// TwinCAT 3 PLC project OC_TwinCAT_EtherCAT
// Title: OC_EtherCAT
// Company: Open Commissioning
// Author: SpiraTec AG
// ProjectVersion: 1.0.0
// Description: Open Commissioning TwinCAT EtherCAT Library
// ProgramVersion: 3.1.4024.0
// libraries:
//   OC_Core, * (Open Commissioning)
//   Tc2_Standard, * (Beckhoff Automation GmbH)
//   Tc2_System, * (Beckhoff Automation GmbH)
//   Tc3_Module, * (Beckhoff Automation GmbH)
//   TcUnit, * (www.tcunit.org)
// project tree:
//   Devices/FB_Beckhoff_EL6001/ E_Beckhoff_EL6001_State.TcDUT (not stored), FB_Beckhoff_EL6001.TcPOU
//   DUTs/ ST_Baumer_Encoder.TcDUT (not stored), ST_Beckhoff_4AI.TcDUT, ST_Beckhoff_2AI.TcDUT, ST_Beckhoff_EL3403.TcDUT, ST_Beckhoff_EL5002.TcDUT, ST_CoE402.TcDUT, ST_Beckhoff_EL9110.TcDUT, ST_Beckhoff_EL9410.TcDUT, ST_Beckhoff_16DI.TcDUT (not stored), ST_Beckhoff_16DO.TcDUT, ST_Beckhoff_4AO.TcDUT (not stored), ST_Beckhoff_4DI_4DO.TcDUT, ST_Beckhoff_8DI.TcDUT (not stored), ST_Beckhoff_8DI_8DO.TcDUT, ST_Beckhoff_8DO.TcDUT, ST_Gefran_GFX4.TcDUT, ST_SEW_SimMovitrac.TcDUT
//   Devices/ FB_Beckhoff_EL5152.TcPOU
//   / PlcTask.TcTTO
//   Tests/Devices/ FB_Beckhoff_EL5152_Test.TcPOU, FB_Beckhoff_EL6001_Test.TcPOU
//   Tests/ PRG_TEST.TcPOU

CONFIGURATION OC_TwinCAT_EtherCAT
    RESOURCE PLC ON TwinCAT3
        TASK PlcTask(INTERVAL := T#1ms, PRIORITY := 30);
        PROGRAM PRG_TEST WITH PlcTask : PRG_TEST;
    END_RESOURCE
END_CONFIGURATION

// ---- DUTs/ST_Beckhoff_4AI.TcDUT
{attribute 'pack_mode' := '1'} 
TYPE ST_Beckhoff_4AI :
STRUCT
	nStatus1	AT %Q* : UINT;
	nValue1		AT %Q* : INT;
	nStatus2	AT %Q* : UINT;
	nValue2		AT %Q* : INT;
END_STRUCT
END_TYPE

// ---- DUTs/ST_Beckhoff_2AI.TcDUT
{attribute 'pack_mode' := '1'} 
TYPE ST_Beckhoff_2AI :
STRUCT
	nStatus1	AT %Q* : UINT;
	nValue1		AT %Q* : INT;
	nStatus2	AT %Q* : UINT;
	nValue2		AT %Q* : INT;
	nStatus3	AT %Q* : UINT;
	nValue3		AT %Q* : INT;
	nStatus4	AT %Q* : UINT;
	nValue4		AT %Q* : INT;
END_STRUCT
END_TYPE

// ---- DUTs/ST_Beckhoff_EL3403.TcDUT
TYPE ST_Beckhoff_EL3403 :
STRUCT
	nCurrent1		AT %Q* : UINT;
	nVoltage1		AT %Q* : UINT;
	nActivePower1	AT %Q* : UINT;
	nCurrent2		AT %Q* : UINT;
	nVoltage2		AT %Q* : UINT;
	nActivePower2	AT %Q* : UINT;	
	nCurrent3		AT %Q* : UINT;
	nVoltage3		AT %Q* : UINT;
	nActivePower3	AT %Q* : UINT;
END_STRUCT
END_TYPE

// ---- DUTs/ST_Beckhoff_EL5002.TcDUT
TYPE ST_Beckhoff_EL5002 :
STRUCT
	nStatus1	AT %Q* : UINT;
	nCounter1	AT %Q* : UDINT;	
	nStatus2	AT %Q* : UINT;
	nCounter2	AT %Q* : UDINT;	
END_STRUCT
END_TYPE

// ---- DUTs/ST_CoE402.TcDUT
{attribute 'pack_mode' := '1'} 
TYPE ST_CoE402 :
STRUCT
	nControlWord	AT %I* : UINT;
	nTargetValue	AT %I* : DINT;
	nStatusWord		AT %Q* : UINT;
	nActualValue	AT %Q* : DINT;
END_STRUCT
END_TYPE

// ---- DUTs/ST_Beckhoff_EL9110.TcDUT
{attribute 'pack_mode' := '1'} 
TYPE ST_Beckhoff_EL9110 :
STRUCT
	bPowerOk	AT %Q* : BIT := TRUE;
END_STRUCT
END_TYPE

// ---- DUTs/ST_Beckhoff_EL9410.TcDUT
{attribute 'pack_mode' := '1'} 
TYPE ST_Beckhoff_EL9410 :
STRUCT
	bUsUndervoltage	AT %Q* : BIT;
	bUpUndervoltage	AT %Q* : BIT;
END_STRUCT
END_TYPE

// ---- DUTs/ST_Beckhoff_16DO.TcDUT
{attribute 'pack_mode' := '1'} 
TYPE ST_Beckhoff_16DO :
STRUCT
	bOut1	AT %I* : BIT;
	bOut2	AT %I* : BIT;
	bOut3	AT %I* : BIT;
	bOut4	AT %I* : BIT;
	bOut5	AT %I* : BIT;
	bOut6	AT %I* : BIT;
	bOut7	AT %I* : BIT;
	bOut8	AT %I* : BIT;
	bOut9	AT %I* : BIT;
	bOut10	AT %I* : BIT;
	bOut11	AT %I* : BIT;
	bOut12	AT %I* : BIT;
	bOut13	AT %I* : BIT;
	bOut14	AT %I* : BIT;
	bOut15	AT %I* : BIT;
	bOut16	AT %I* : BIT;
END_STRUCT
END_TYPE

// ---- DUTs/ST_Beckhoff_4DI_4DO.TcDUT
{attribute 'pack_mode' := '1'} 
TYPE ST_Beckhoff_4DI_4DO :
STRUCT
	bIn1	AT %Q* : BIT;
	bIn2	AT %Q* : BIT;
	bIn3	AT %Q* : BIT;
	bIn4	AT %Q* : BIT;	
	bOut1	AT %I* : BIT;
	bOut2	AT %I* : BIT;
	bOut3	AT %I* : BIT;
	bOut4	AT %I* : BIT;	
END_STRUCT
END_TYPE

// ---- DUTs/ST_Beckhoff_8DI_8DO.TcDUT
{attribute 'pack_mode' := '1'} 
TYPE ST_Beckhoff_8DI_8DO :
STRUCT
	bIn1	AT %Q* : BIT;
	bIn2	AT %Q* : BIT;
	bIn3	AT %Q* : BIT;
	bIn4	AT %Q* : BIT;
	bIn5	AT %Q* : BIT;
	bIn6	AT %Q* : BIT;
	bIn7	AT %Q* : BIT;
	bIn8	AT %Q* : BIT;
	bOut1	AT %I* : BIT;
	bOut2	AT %I* : BIT;
	bOut3	AT %I* : BIT;
	bOut4	AT %I* : BIT;
	bOut5	AT %I* : BIT;
	bOut6	AT %I* : BIT;
	bOut7	AT %I* : BIT;
	bOut8	AT %I* : BIT;
END_STRUCT
END_TYPE

// ---- DUTs/ST_Beckhoff_8DO.TcDUT
{attribute 'pack_mode' := '1'} 
TYPE ST_Beckhoff_8DO :
STRUCT
	bOut1	AT %I* : BIT;
	bOut2	AT %I* : BIT;
	bOut3	AT %I* : BIT;
	bOut4	AT %I* : BIT;
	bOut5	AT %I* : BIT;
	bOut6	AT %I* : BIT;
	bOut7	AT %I* : BIT;
	bOut8	AT %I* : BIT;
END_STRUCT
END_TYPE

// ---- DUTs/ST_Gefran_GFX4.TcDUT
{attribute 'pack_mode' := '1'} 
TYPE ST_Gefran_GFX4 :
STRUCT
	nProcessVariable1	AT %Q* : INT;
	nControllerStatus1	AT %Q* : UINT;	
	nOutputPower1		AT %Q* : INT;
	nProcessVariable2	AT %Q* : INT;
	nControllerStatus2	AT %Q* : UINT;	
	nOutputPower2		AT %Q* : INT;
	nProcessVariable3	AT %Q* : INT;
	nControllerStatus3	AT %Q* : UINT;	
	nOutputPower3		AT %Q* : INT;
	nProcessVariable4	AT %Q* : INT;
	nControllerStatus4	AT %Q* : UINT;	
	nOutputPower4		AT %Q* : INT;
	nLocalSetpoint1		AT %I* : INT;
	nLocalSetpoint2		AT %I* : INT;
	nLocalSetpoint3		AT %I* : INT;
	nLocalSetpoint4		AT %I* : INT;
END_STRUCT
END_TYPE

// ---- DUTs/ST_SEW_SimMovitrac.TcDUT
{attribute 'pack_mode' := '1'}
TYPE ST_SEW_SimMovitrac :
STRUCT
	PI1		AT %Q* : WORD;
	PI2		AT %Q* : WORD;
	PI3		AT %Q* : WORD;
	PO1		AT %I* : WORD;
	PO2		AT %I* : WORD;
	PO3		AT %I* : WORD;
END_STRUCT
END_TYPE

// ---- Tests/PRG_TEST.TcPOU
PROGRAM PRG_TEST
VAR	
	FB_System	: FB_System;
	FB_Beckhoff_EL5152_Test : FB_Beckhoff_EL5152_Test;
	FB_Beckhoff_EL6001_Test : FB_Beckhoff_EL6001_Test;
	FB_DS402_FSM_Test : FB_DS402_FSM_Test;	
	FB_DS402_CSP_Test : FB_DS402_CSP_Test; 
	FB_Sercos_FSM_Test : FB_Sercos_FSM_Test;
	FB_Sercos_VC_Test : FB_Sercos_VC_Test;
END_VAR

FB_System();
TcUnit.RUN();

END_PROGRAM

// ---- Tests/Devices/FB_Beckhoff_EL5152_Test.TcPOU
FUNCTION_BLOCK FB_Beckhoff_EL5152_Test EXTENDS TcUnit.FB_TestSuite
VAR
	fbDevice : FB_Beckhoff_EL5152;
	nExpected : UINT;
	nResult : UINT;
END_VAR

TEST('nCounter1');
nExpected := 111;
fbDevice.nValue1 := nExpected;
fbDevice();
nResult := fbDevice.Counter1;
AssertEquals(Expected := nExpected,
             Actual := nResult,
             Message := 'nCounter1 value is not correct');	
TEST_FINISHED();

TEST('nCounter2');
nExpected := 112;
fbDevice.nValue2 := nExpected;
fbDevice();
nResult := fbDevice.Counter2;
AssertEquals(Expected := nExpected,
             Actual := nResult,
             Message := 'nCounter2 value is not correct');	
TEST_FINISHED();


TEST('nStatus1');
nExpected := 4;
fbDevice.Control1 := nExpected;
fbDevice();
nResult := fbDevice.Status1;
AssertEquals(Expected := nExpected,
             Actual := nResult,
             Message := 'nStatus1 value is not correct');	
TEST_FINISHED();

TEST('nStatus2');
nExpected := 4;
fbDevice.Control2 := nExpected;
fbDevice();
nResult := fbDevice.Status2;
AssertEquals(Expected := nExpected,
             Actual := nResult,
             Message := 'nStatus2 value is not correct');	
TEST_FINISHED();

END_FUNCTION_BLOCK

// ---- Devices/FB_Beckhoff_EL5152.TcPOU
FUNCTION_BLOCK FB_Beckhoff_EL5152
VAR_INPUT
	nValue1		: UINT;
	nValue2		: UINT;
END_VAR
VAR_OUTPUT
END_VAR
VAR
	nControl1		AT %I* : UINT;
	nSetCounter1	AT %I* : UINT;
	nControl2		AT %I* : UINT;
	nSetCounter2	AT %I* : UINT;
	
	nStatus1		AT %Q* : UINT;
	nCounter1		AT %Q* : UINT;	
	nPeriod1    	AT %Q* : UDINT;
	nStatus2		AT %Q* : UINT;
	nCounter2		AT %Q* : UINT;
	nPeriod2    	AT %Q* : UDINT;
END_VAR

nStatus1.2 := nControl1.2;
nStatus2.2 := nControl2.2;

nCounter1 := nValue1;
nCounter2 := nValue2;

END_FUNCTION_BLOCK

// ---- Tests/Devices/FB_Beckhoff_EL6001_Test.TcPOU
FUNCTION_BLOCK FB_Beckhoff_EL6001_Test EXTENDS TcUnit.FB_TestSuite
VAR
	fbDevice : FB_Beckhoff_EL6001;
	nExpected : UINT;
	nResult : UINT;
END_VAR

TestProperties();
TestState();

METHOD TestProperties : REFERENCE TO FB_Test
VAR
	bExpected 		: BOOL;
	bResult 		: BOOL;
END_VAR
TEST('TransmitRequest FALSE');
bExpected := FALSE; 
fbDevice();
fbDevice.Control := 0;
fbDevice();
bResult := fbDevice.TransmitRequest;
AssertEquals(Expected := bExpected,
             Actual := bResult,
             Message := 'TransmitRequest value is not correct');		
TEST_FINISHED();

TEST('TransmitRequest TRUE');
bExpected := TRUE; 
fbDevice();
fbDevice.Control := 1;
fbDevice();
bResult := fbDevice.TransmitRequest;
AssertEquals(Expected := bExpected,
             Actual := bResult,
             Message := 'TransmitRequest value is not correct');		
TEST_FINISHED();

TEST('ReceiveAccepted FALSE');
bExpected := FALSE; 
fbDevice();
fbDevice.Control := 0;
fbDevice();
bResult := fbDevice.ReceiveAccepted;
AssertEquals(Expected := bExpected,
             Actual := bResult,
             Message := 'ReceiveAccepted value is not correct');		
TEST_FINISHED();

TEST('ReceiveAccepted TRUE');
bExpected := TRUE; 
fbDevice();
fbDevice.Control := 2;
fbDevice();
bResult := fbDevice.ReceiveAccepted;
AssertEquals(Expected := bExpected,
             Actual := bResult,
             Message := 'ReceiveAccepted value is not correct');		
TEST_FINISHED();

TEST('InitRequest TRUE');
bExpected := TRUE; 
fbDevice();
fbDevice.Control := 4;
fbDevice();
bResult := fbDevice.InitRequest;
AssertEquals(Expected := bExpected,
             Actual := bResult,
             Message := 'InitRequest value is not correct');		
TEST_FINISHED();

TEST('SendContinuous TRUE');
bExpected := TRUE; 
fbDevice.Control := 0;
fbDevice();
fbDevice.Control := 9;
fbDevice();
bResult := fbDevice.SendContinuous;
AssertEquals(Expected := bExpected,
             Actual := bResult,
             Message := 'SendContinuous value is not correct');		
TEST_FINISHED();
END_METHOD

METHOD TestState : REFERENCE TO FB_Test
VAR
	bResult 		: BOOL;
	nDataSend 		:  ARRAY[0..50] OF BYTE;
END_VAR
TEST('Transition: INIT - READY');
fbDevice.Control := 0;
fbDevice.State := E_Beckhoff_EL6001_State.INIT;	
fbDevice();

AssertTRUE(fbDevice.State = E_Beckhoff_EL6001_State.READY, 'State value is not correct');
	
TEST_FINISHED();

TEST('Transition: READY - TRANSMIT');
fbDevice.Control := 0;
fbDevice.State := E_Beckhoff_EL6001_State.READY;	
fbDevice();

fbDevice.Control := 257;
fbDevice();

AssertTRUE(fbDevice.State = E_Beckhoff_EL6001_State.TRANSMIT, 'State value is not correct');
	
TEST_FINISHED();

TEST('Transition: READY - RECEIVE');
fbDevice.Control := 0;
fbDevice.State := E_Beckhoff_EL6001_State.READY;	
fbDevice();

fbDevice.bSend := TRUE;
fbDevice.pDataIn := ADR(nDataSend);
fbDevice.nLength := 1;
fbDevice.Control := 1;
fbDevice();

fbDevice.bSend := FALSE;
fbDevice.nLength := 0;

AssertTRUE(fbDevice.State = E_Beckhoff_EL6001_State.RECEIVE, 'State value is not correct');
TEST_FINISHED();
END_METHOD

END_FUNCTION_BLOCK

// ---- Devices/FB_Beckhoff_EL6001/FB_Beckhoff_EL6001.TcPOU
FUNCTION_BLOCK FB_Beckhoff_EL6001
VAR_INPUT
	bSend				: BOOL;
	nLength				: UINT;
	pDataIn				: POINTER TO BYTE; //Data to send
	pDataOut			: POINTER TO BYTE; //Received data when nDataAvailable > 0.
END_VAR
VAR_OUTPUT
	bBusy				: BOOL;
	nDataAvailable		: INT; //Received bytes. Only available for one cycle.
END_VAR
VAR
	nControl			AT %I* : UINT;
	nDataOut			AT %I* : ARRAY[0..21] OF USINT;
	nStatus				AT %Q* : UINT;
	nDataIn				AT %Q* : ARRAY[0..21] OF USINT;
END_VAR
VAR
	nControlByte		: BYTE;
	nOutLength			: BYTE;	
	bTransmitRequest	: BOOL;
	bReceiveAccecpted	: BOOL;
	bInitRequest		: BOOL;
	bSendContinuous		: BOOL;
	
	bTransmitAccepted	: BOOL;
	bReceiveRequest		: BOOL;
	bInitAccepted		: BOOL;
	bBufferFull			: BOOL;
	bParityError		: BOOL;
	bFramingError		: BOOL;
	bOverrunError		: BOOL;
	nInLength			: BYTE;
	
	nPendingLength		: UINT;
	nOffsetNext			: UINT;
	
	eState				: E_Beckhoff_EL6001_State;
	trigSend			: R_TRIG;
END_VAR

(* Receive control word *)
	bTransmitRequest 	:= nControl.0 <> nControlByte.0;
	bReceiveAccecpted 	:= nControl.1 <> nControlByte.1;
	bInitRequest		:= nControl = 4;
	bSendContinuous		:= nControl.3 AND NOT nControlByte.0;	
	nControlByte 		:= F_GetLByte(nControl);
	nOutLength 			:= F_GetHByte(nControl);

(* Initialize *)
	IF bInitRequest THEN
		eState := E_Beckhoff_EL6001_State.INIT;			
	END_IF
	
CASE eState OF
	E_Beckhoff_EL6001_State.INIT:
		bTransmitAccepted 	:= FALSE;
		bReceiveRequest		:= FALSE;
		bInitAccepted		:= TRUE;
		bBufferFull			:= FALSE;
		bParityError		:= FALSE;
		bFramingError		:= FALSE;
		bOverrunError		:= FALSE;
		nInLength			:= 0;
		nDataAvailable		:= 0;
		
		// -> INIT_READY
		IF nControl = 0 THEN
			bInitAccepted := FALSE;		
			eState := E_Beckhoff_EL6001_State.READY;
		END_IF

	E_Beckhoff_EL6001_State.READY:
		nDataAvailable := 0;

		// -> TRANSMIT
		IF bTransmitRequest AND nOutLength > 0 AND nOutLength < 23 THEN
			eState := E_Beckhoff_EL6001_State.TRANSMIT;
			RETURN;
		END_IF
		
		trigSend(CLK := bSend);
		
		// -> RECEIVE
		IF trigSend.Q AND nLength > 0 AND pDataIn <> 0 THEN
			bReceiveRequest := NOT bReceiveRequest;
			nPendingLength := nLength;
			nInLength := UINT_TO_BYTE(MIN(22, nPendingLength));
			memcpy(ADR(nDataIn), pDataIn, nInLength);		
			eState := E_Beckhoff_EL6001_State.RECEIVE;
		END_IF	
		
	E_Beckhoff_EL6001_State.TRANSMIT:
		IF pDataOut <> 0 THEN
			memcpy(pDataOut, ADR(nDataOut), nOutLength);
		END_IF
		bTransmitAccepted := NOT bTransmitAccepted;
		nDataAvailable := nOutLength;
		eState := E_Beckhoff_EL6001_State.READY;
		
	E_Beckhoff_EL6001_State.RECEIVE:
		IF bReceiveAccecpted THEN
			nOffsetNext := nInLength;
			nPendingLength := nPendingLength - nOffsetNext;
			IF nPendingLength = 0 THEN
				eState := E_Beckhoff_EL6001_State.READY;
			END_IF
			IF nPendingLength > 0 THEN
				bReceiveRequest := NOT bReceiveRequest;
				nInLength := UINT_TO_BYTE(MIN(22, nPendingLength));
				memcpy(ADR(nDataIn), pDataIn + nOffsetNext, nInLength);
				eState := E_Beckhoff_EL6001_State.RECEIVE;
			END_IF				
		END_IF
	
END_CASE

bBusy := eState <> E_Beckhoff_EL6001_State.READY;
	
(* Send status word *)
	nStatus.0			:= bTransmitAccepted;
	nStatus.1			:= bReceiveRequest;
	nStatus.2			:= bInitAccepted;
	nStatus.3			:= bBufferFull;
	nStatus.4			:= bParityError;
	nStatus.5			:= bFramingError;
	nStatus.6			:= bOverrunError;
	memcpy(ADR(nStatus) + 1, ADR(nInLength), 1);

PROPERTY INTERNAL BufferFull : BOOl
GET
BufferFull := bBufferFull;
END_GET
END_PROPERTY

PROPERTY INTERNAL Control : UINT
SET
nControl := Control;
END_SET
END_PROPERTY

PROPERTY INTERNAL FramingError : BOOl
GET
FramingError := bFramingError;
END_GET
END_PROPERTY

PROPERTY INTERNAL InitAccepted : BOOl
GET
InitAccepted := bInitAccepted;
END_GET
END_PROPERTY

PROPERTY INTERNAL InitRequest : BOOl
GET
InitRequest := bInitRequest;
END_GET
END_PROPERTY

PROPERTY INTERNAL OverrunError : BOOl
GET
OverrunError := bOverrunError;
END_GET
END_PROPERTY

PROPERTY INTERNAL ParityError : BOOl
GET
ParityError := bParityError;
END_GET
END_PROPERTY

PROPERTY INTERNAL ReceiveAccepted : BOOl
GET
ReceiveAccepted := bReceiveAccecpted;
END_GET
END_PROPERTY

PROPERTY INTERNAL ReceiveRequest : BOOl
GET
ReceiveRequest := bReceiveRequest;
END_GET
END_PROPERTY

PROPERTY INTERNAL SendContinuous : BOOl
GET
SendContinuous := bSendContinuous;
END_GET
END_PROPERTY

PROPERTY INTERNAL State : E_Beckhoff_EL6001_State
GET
State := eState;
END_GET
SET
eState := State;
END_SET
END_PROPERTY

PROPERTY INTERNAL TransmitAccepted : BOOl
GET
TransmitAccepted := bTransmitAccepted;
END_GET
END_PROPERTY

PROPERTY INTERNAL TransmitRequest : BOOl
GET
TransmitRequest := bTransmitRequest;
END_GET
END_PROPERTY

END_FUNCTION_BLOCK
